TYPE T_PositiveINT : INT(0..32767); END_TYPE

(* stored: Version 1.1.0.1
   DUT T_PositiveINT: Id {b43a706f-755f-49b6-ab99-f15014041a46} *)
